INTERFACE I_Middleware

METHOD Handle
VAR_INPUT
	Request : I_Request;
	Response : I_ServerResponse;
END_VAR
END_METHOD

PROPERTY PUBLIC NextMiddleware : I_Middleware
GET
END_GET
SET
END_SET
END_PROPERTY

END_INTERFACE

(* stored: Version 1.1.0.1, ProductVersion 3.1.4026.13
   Itf I_Middleware: Id {c6de0511-8791-47bc-bd05-1e7ea8dec882}
   Method Handle: Id {e9ed1e8e-e1ba-4a07-b915-3a53a228db40}
   Property NextMiddleware: Id {d4daed27-77d0-4d8e-a40c-7c2ca31b310d}
   Get Get: Id {c4f5edea-4997-466e-a8e1-409427ed23e4}
   Set Set: Id {73f564f5-34fe-4e43-9705-8b982564aae5} *)
